FUNCTION "_alarmBit01Id" : Void
TITLE = Function:Update alarm ID, check 1 bit
{ S7_Optimized_Access := 'TRUE' }
AUTHOR : cyanezf
FAMILY : Alarm
NAME : _alarmBit01Id
VERSION : 1.0

   VAR_INPUT
      triggered : Bool;   // 1=Some alarm in controller alarm group
      a00 : Bool;   // 1=Alarm
      a00_id : Int;   // 0=No ID; 0xHHHH=Some alarm ID
   END_VAR

   VAR_IN_OUT
      id : Int; // Alarm id variable in controller alarm group
   END_VAR

   VAR CONSTANT
      NO_ALARM : Int := 0;
   END_VAR

BEGIN
	(*--{
		"Log": [
			{"version":"v1.0", "date" : "2025-01-27", "author": "cyanezf, "description": "First version"},
		],
		"dependencies" : [],
		"description" : "

How it works:
Alarm #id is set with #a00_id when #a00 is true and #id is equal to #NO_ALARM
Alarm #id is set with #NO_ALARM when #triggered is false;
	 "
	}--*)

	// Clear if not triggered
	IF NOT #triggered THEN
	  #id := #NO_ALARM;
	  ENO := true;
		RETURN;
	end_if;

	// Check alarm
	IF #a00 THEN
	  IF #id = #NO_ALARM THEN
	    #id := #a00_id;
	    ENO := true;
	    RETURN;
	  END_IF;

	ELSE
	  IF #id = #a00_id THEN
	    #id := #NO_ALARM;
	  END_IF;
	END_IF;

	// Save RLO
	ENO := true;

END_FUNCTION

